TYPE U_TOUCH_PROBE_STATE :
UNION
  stState              : ARRAY[1..MAX_TOUCH_PROBE] OF ST_STATE_TOUCH_PROBE;

  byState    AT %Q*   : ARRAY[1..MAX_TOUCH_PROBE] OF
                        ARRAY[1..SIZEOF(ST_STATE_TOUCH_PROBE)] OF BYTE;
END_UNION
END_TYPE

(* stored: Version 1.1.0.1, ProductVersion 3.1.4026.13
   DUT U_TOUCH_PROBE_STATE: Id {71c7ab25-1174-46f1-a5db-0c3a22dfe6c9} *)
